{attribute 'strict'}
{attribute 'to_string'}
TYPE E_SystemState :
(
    INIT             := 0,
    HOMING_REQUIRED  := 1,
    READY            := 2,
    RUN              := 3,
    FAULT            := 4
);
END_TYPE

(* stored: Version 1.1.0.1, ProductVersion 3.1.4026.18
   DUT E_SystemState: Id {9f958ac8-f1c4-4fa6-a7fa-32a7593fcb5d} *)
